// TwinCAT 3 PLC project PLC
// ProgramVersion: 3.1.4024.0
// libraries:
//   Tc2_Standard, * (Beckhoff Automation GmbH)
//   Tc2_System, * (Beckhoff Automation GmbH)
//   Tc3_Module, * (Beckhoff Automation GmbH)
// project tree:
//   / PlcTask.TcTTO
//   POUs/ MAIN.TcPOU
// real-time tasks:
//   TASK PlcTask: cycle T#10ms, priority 20, ADS port 350

CONFIGURATION PLC
    RESOURCE PLC ON TwinCAT3
        TASK PlcTask(INTERVAL := T#10ms, PRIORITY := 20);
        PROGRAM MAIN WITH PlcTask : MAIN;
    END_RESOURCE
END_CONFIGURATION

// ---- POUs/MAIN.TcPOU
PROGRAM MAIN
VAR
	Sensor1: BOOL;
	Sensor2: BOOL;
	Sensor3: BOOL;
	

	Motor1: BOOL;
	Motor2: BOOL;
	Motor3: BOOL;
	
	Sensor1On: BOOL;
	tonM2: TON;
	tonM1: TON;


END_VAR

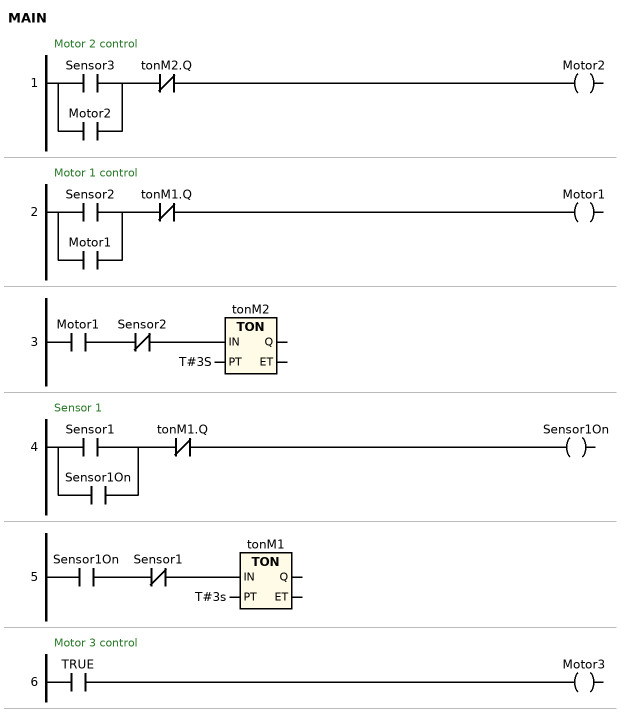
// NETWORK 1
// Motor 2 control
Motor2 := (Sensor3 OR Motor2) AND NOT tonM2.Q;

// NETWORK 2
// Motor 1 control
Motor1 := (Sensor2 OR Motor1) AND NOT tonM1.Q;

// NETWORK 3
tonM2(IN := Motor1 AND NOT Sensor2, PT := T#3S); // TON

// NETWORK 4
// Sensor 1
Sensor1On := (Sensor1 OR Sensor1On) AND NOT tonM1.Q;

// NETWORK 5
tonM1(IN := Sensor1On AND NOT Sensor1, PT := T#3s); // TON

// NETWORK 6
// Motor 3 control
Motor3 := TRUE;

END_PROGRAM
